Universal Robots PolyScope program: reciprocal_full.urp

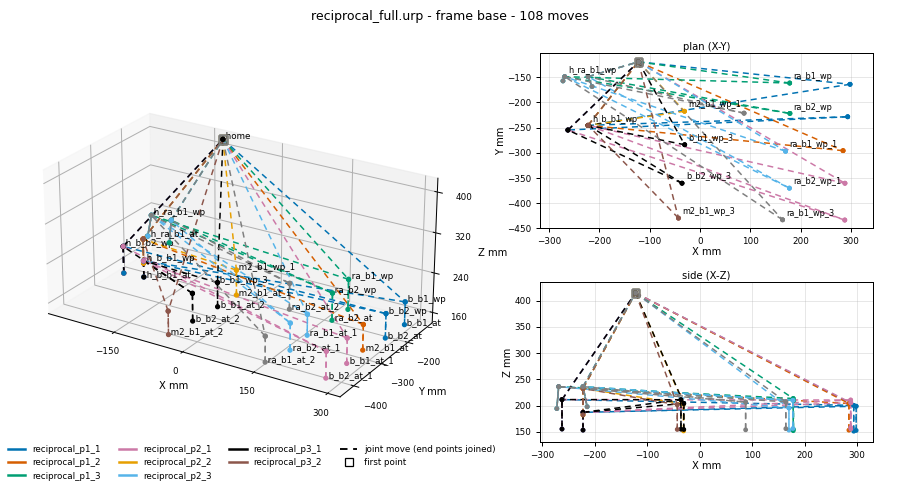
[picture p0: tool path of reciprocal_full.urp in frame base, 108 of 108 moves have a stored position in this frame; points joined in program order, loops and branches not executed]
Program reciprocal_full (installation=default directory=/programs/ITER createdIn=5.3.1.64192 lastSavedIn=5.3.1.64192 robotSerialNumber=20195300365)
Calibrated DH parameters: a=[-0.000093, -0.190649, -0.212673, 0.000091, -0.000205, 0]; d=[0.151591, 44.061648, -42.488068, -1.442789, 0.085322, 0.091911]; alpha=[1.570082, -0.003447, 0.007513, 1.572293, -1.571904, 0]; deltaTheta=[0, -0.672656, 0.728185, -0.055522, 0.000005, 0]
Robot Program (runOnlyOnce=true)
  Call reciprocal_p1_1
  Popup Message (haltProgram=false message=interaction inputType=Text)
  Call reciprocal_p1_2
  Popup Message (haltProgram=false message=interaction inputType=Text)
  Call reciprocal_p1_3
  Popup Message (haltProgram=false message=interaction inputType=Text)
  Call reciprocal_p2_1
  Popup Message (haltProgram=false message=interaction inputType=Text)
  Call reciprocal_p2_2
  Popup Message (haltProgram=false message=interaction inputType=Text)
  Call reciprocal_p2_3
  Popup Message (haltProgram=false message=interaction inputType=Text)
  Call reciprocal_p3_1
  Popup Message (haltProgram=false message=interaction inputType=Text)
  Call reciprocal_p3_2
  Popup Message (haltProgram=false message=interaction inputType=Text)
  Call reciprocal_p3_3
SubProgram -> reciprocal_p3_3
SubProgram -> reciprocal_p3_2
SubProgram -> reciprocal_p3_1
SubProgram -> reciprocal_p2_3
SubProgram -> reciprocal_p2_2
SubProgram -> reciprocal_p2_1
SubProgram -> reciprocal_p1_3
SubProgram -> reciprocal_p1_2
SubProgram -> reciprocal_p1_1
SubProgram reciprocal_p1_1 (keepSynchronizedWithDisk=true trackProgramExecution=false) programFile=/programs/ITER/reciprocal_p1_1.urp
  URCap Gripper Activate (Robotiq_Grippers, Robotiq Inc.) dataModel(ResetAndActivateKey=false)
  URCap Gripper (Robotiq_Grippers, Robotiq Inc.) dataModel(position=50.0, force=100.0, speed=100.0, positionInDouble=50.0, forceInDouble=100.0, speedInDouble=100.0, slaveIds=[9], blocking=true)
  MoveJ speed 60 deg/s, acceleration 80 deg/s^2 (useActiveTCP=true) feature=Base
    Waypoint home: TCP in base x=-122.15 y=-119.32 z=414.454 mm, rx=2.2563 ry=2.1459 rz=-0.0481 rad; joints [-85.681, -56.776, -79.802, -131.025, 89.944, -262.833] deg
  Folder Base
    MoveJ speed 60 deg/s, acceleration 80 deg/s^2 (useActiveTCP=true) feature=Base
      Waypoint b_b1_wp: TCP in base x=297.989 y=-163.874 z=198.695 mm, rx=2.2416 ry=2.1933 rz=-0.0875 rad; joints [-5.657, -99.775, -108.03, -64.017, 87.69, -183.98] deg
      Waypoint b_b1_at: TCP in base x=297.98 y=-163.89 z=152.63 mm, rx=2.2418 ry=2.1932 rz=-0.0874 rad; joints [-5.678, -106.278, -114.473, -51.073, 87.63, -183.927] deg
      URCap Gripper (Robotiq_Grippers, Robotiq Inc.) dataModel(position=100.0, force=100.0, speed=100.0, positionInDouble=100.0, forceInDouble=100.0, speedInDouble=100.0, slaveIds=[9], blocking=true)
      Waypoint b_b1_wp: TCP in base x=297.989 y=-163.874 z=198.695 mm, rx=2.2416 ry=2.1933 rz=-0.0875 rad; joints [-5.657, -99.775, -108.03, -64.017, 87.69, -183.98] deg
      Waypoint h_b_b1_wp: TCP in base x=-222.187 y=-245.349 z=187.06 mm, rx=-3.1315 ry=0.0204 rz=0.0123 rad; joints [-108.957, -99.116, -113.081, -58.146, 89.665, -197.782] deg
      Waypoint h_b_b1_at: TCP in base x=-222.188 y=-245.348 z=153.24 mm, rx=-3.1314 ry=0.0204 rz=0.0122 rad; joints [-108.969, -104.391, -117.643, -48.312, 89.612, -197.745] deg
      URCap Gripper (Robotiq_Grippers, Robotiq Inc.) dataModel(position=50.0, force=100.0, speed=100.0, positionInDouble=50.0, forceInDouble=100.0, speedInDouble=100.0, slaveIds=[9], blocking=true)
      Waypoint h_b_b1_wp: TCP in base x=-222.187 y=-245.349 z=187.06 mm, rx=-3.1315 ry=0.0204 rz=0.0123 rad; joints [-108.957, -99.116, -113.081, -58.146, 89.665, -197.782] deg
    MoveJ speed 60 deg/s, acceleration 80 deg/s^2 (useActiveTCP=true) feature=Base
      Waypoint b_b2_wp: TCP in base x=293.357 y=-228.364 z=200.348 mm, rx=2.2516 ry=2.1757 rz=-0.0473 rad; joints [-17.02, -106.79, -99.111, -64.372, 88.479, -194.689] deg
      Waypoint b_b2_at: TCP in base x=293.371 y=-228.346 z=151.163 mm, rx=2.2516 ry=2.1757 rz=-0.0473 rad; joints [-17.033, -113.072, -105.562, -51.642, 88.423, -194.639] deg
      URCap Gripper (Robotiq_Grippers, Robotiq Inc.) dataModel(position=100.0, force=100.0, speed=100.0, positionInDouble=100.0, forceInDouble=100.0, speedInDouble=100.0, slaveIds=[9], blocking=true)
      Waypoint b_b2_wp: TCP in base x=293.357 y=-228.364 z=200.348 mm, rx=2.2516 ry=2.1757 rz=-0.0473 rad; joints [-17.02, -106.79, -99.111, -64.372, 88.479, -194.689] deg
      Waypoint h_b_b2_wp: TCP in base x=-262.196 y=-254.726 z=211.351 mm, rx=-3.0605 ry=0.0443 rz=-0.0223 rad; joints [-114.749, -105.359, -96.042, -73.109, 89.199, -202.734] deg
      Waypoint h_b_b2_at: TCP in base x=-262.208 y=-254.718 z=155.33 mm, rx=-3.0605 ry=0.0443 rz=-0.0223 rad; joints [-114.774, -111.736, -104.192, -58.581, 89.146, -202.674] deg
      URCap Gripper (Robotiq_Grippers, Robotiq Inc.) dataModel(position=50.0, force=100.0, speed=100.0, positionInDouble=50.0, forceInDouble=100.0, speedInDouble=100.0, slaveIds=[9], blocking=true)
      Waypoint h_b_b2_wp: TCP in base x=-262.196 y=-254.726 z=211.351 mm, rx=-3.0605 ry=0.0443 rz=-0.0223 rad; joints [-114.749, -105.359, -96.042, -73.109, 89.199, -202.734] deg
  MoveJ speed 60 deg/s, acceleration 80 deg/s^2 (useActiveTCP=true) feature=Base
    Waypoint home: TCP in base x=-122.15 y=-119.32 z=414.454 mm, rx=2.2563 ry=2.1459 rz=-0.0481 rad; joints [-85.681, -56.776, -79.802, -131.025, 89.944, -262.833] deg
SubProgram reciprocal_p1_2 (keepSynchronizedWithDisk=true trackProgramExecution=false) programFile=/programs/ITER/reciprocal_p1_2.urp
  URCap Gripper Activate (Robotiq_Grippers, Robotiq Inc.) dataModel(ResetAndActivateKey=false)
  URCap Gripper (Robotiq_Grippers, Robotiq Inc.) dataModel(position=50.0, force=100.0, speed=100.0, positionInDouble=50.0, forceInDouble=100.0, speedInDouble=100.0, slaveIds=[9], blocking=true)
  MoveJ speed 60 deg/s, acceleration 80 deg/s^2 (useActiveTCP=true) feature=Base
    Waypoint home: TCP in base x=-122.15 y=-119.32 z=414.454 mm, rx=2.2563 ry=2.1459 rz=-0.0481 rad; joints [-85.681, -56.776, -79.802, -131.025, 89.944, -262.833] deg
  Folder Mid_2
    MoveJ speed 60 deg/s, acceleration 80 deg/s^2 (useActiveTCP=true) feature=Base
      Waypoint m2_b1_wp: TCP in base x=284.16 y=-295.685 z=203.947 mm, rx=2.2476 ry=2.1381 rz=-0.0269 rad; joints [-27.296, -114.823, -87.386, -65.934, 88.586, -204.141] deg
      Waypoint m2_b1_at: TCP in base x=284.146 y=-295.69 z=153.108 mm, rx=2.2477 ry=2.1381 rz=-0.0269 rad; joints [-27.314, -120.451, -93.885, -53.812, 88.539, -204.094] deg
      URCap Gripper (Robotiq_Grippers, Robotiq Inc.) dataModel(position=100.0, force=100.0, speed=100.0, positionInDouble=100.0, forceInDouble=100.0, speedInDouble=100.0, slaveIds=[9], blocking=true)
      Waypoint m2_b1_wp: TCP in base x=284.16 y=-295.685 z=203.947 mm, rx=2.2476 ry=2.1381 rz=-0.0269 rad; joints [-27.296, -114.823, -87.386, -65.934, 88.586, -204.141] deg
      Waypoint h_m2_b1_wp: TCP in base x=-222.193 y=-245.34 z=232.403 mm, rx=-3.1314 ry=0.0205 rz=0.0123 rad; joints [-108.936, -94.247, -105.13, -70.966, 89.712, -197.837] deg
      Waypoint h_m2_b1_at: TCP in base x=-222.194 y=-245.343 z=182.32 mm, rx=-3.1314 ry=0.0205 rz=0.0122 rad; joints [-108.96, -99.771, -113.792, -56.782, 89.658, -197.776] deg
      URCap Gripper (Robotiq_Grippers, Robotiq Inc.) dataModel(position=50.0, force=100.0, speed=100.0, positionInDouble=50.0, forceInDouble=100.0, speedInDouble=100.0, slaveIds=[9], blocking=true)
      Waypoint h_m2_b1_wp: TCP in base x=-222.193 y=-245.34 z=232.403 mm, rx=-3.1314 ry=0.0205 rz=0.0123 rad; joints [-108.936, -94.247, -105.13, -70.966, 89.712, -197.837] deg
  MoveJ speed 60 deg/s, acceleration 80 deg/s^2 (useActiveTCP=true) feature=Base
    Waypoint home: TCP in base x=-122.15 y=-119.32 z=414.454 mm, rx=2.2563 ry=2.1459 rz=-0.0481 rad; joints [-85.681, -56.776, -79.802, -131.025, 89.944, -262.833] deg
SubProgram reciprocal_p1_3 (keepSynchronizedWithDisk=true trackProgramExecution=false) programFile=/programs/ITER/reciprocal_p1_3.urp
  URCap Gripper Activate (Robotiq_Grippers, Robotiq Inc.) dataModel(ResetAndActivateKey=false)
  URCap Gripper (Robotiq_Grippers, Robotiq Inc.) dataModel(position=50.0, force=100.0, speed=100.0, positionInDouble=50.0, forceInDouble=100.0, speedInDouble=100.0, slaveIds=[9], blocking=true)
  MoveJ speed 60 deg/s, acceleration 80 deg/s^2 (useActiveTCP=true) feature=Base
    Waypoint home: TCP in base x=-122.15 y=-119.32 z=414.454 mm, rx=2.2563 ry=2.1459 rz=-0.0481 rad; joints [-85.681, -56.776, -79.802, -131.025, 89.944, -262.833] deg
  Folder Roof_A
    MoveJ speed 60 deg/s, acceleration 80 deg/s^2 (useActiveTCP=true) feature=Base
      Waypoint ra_b1_wp: TCP in base x=178.147 y=-161.416 z=213.493 mm, rx=2.2107 ry=2.1864 rz=-0.0129 rad; joints [-8.931, -69.528, -131.792, -67.419, 88.9, -187.899] deg
      Waypoint ra_b1_at: TCP in base x=178.14 y=-161.425 z=152.15 mm, rx=2.2108 ry=2.1863 rz=-0.013 rad; joints [-8.971, -81.208, -143.947, -43.587, 88.771, -187.8] deg
      URCap Gripper (Robotiq_Grippers, Robotiq Inc.) dataModel(position=100.0, force=100.0, speed=100.0, positionInDouble=100.0, forceInDouble=100.0, speedInDouble=100.0, slaveIds=[9], blocking=true)
      Waypoint ra_b1_wp: TCP in base x=178.147 y=-161.416 z=213.493 mm, rx=2.2107 ry=2.1864 rz=-0.0129 rad; joints [-8.931, -69.528, -131.792, -67.419, 88.9, -187.899] deg
      Waypoint h_ra_b1_wp: TCP in base x=-268.55 y=-148.787 z=236.04 mm, rx=2.7608 ry=-0.1306 rz=0.0749 rad; joints [-131.096, -88.368, -118.927, -47.1, 105.838, -213.026] deg
      Waypoint h_ra_b1_at: TCP in base x=-272.048 y=-157.193 z=194.251 mm, rx=2.7928 ry=-0.086 rz=0.1068 rad; joints [-130.55, -96.287, -122.586, -37.872, 105.802, -214.66] deg
      URCap Gripper (Robotiq_Grippers, Robotiq Inc.) dataModel(position=50.0, force=100.0, speed=100.0, positionInDouble=50.0, forceInDouble=100.0, speedInDouble=100.0, slaveIds=[9], blocking=true)
      Waypoint h_ra_b1_wp: TCP in base x=-268.55 y=-148.787 z=236.04 mm, rx=2.7608 ry=-0.1306 rz=0.0749 rad; joints [-131.096, -88.368, -118.927, -47.1, 105.838, -213.026] deg
    MoveJ speed 60 deg/s, acceleration 80 deg/s^2 (useActiveTCP=true) feature=Base
      Waypoint ra_b2_wp: TCP in base x=178.587 y=-221.707 z=209.682 mm, rx=2.2093 ry=2.1872 rz=-0.0611 rad; joints [-23.097, -83.646, -122.705, -62.748, 87.545, -202.118] deg
      Waypoint ra_b2_at: TCP in base x=178.563 y=-221.705 z=154.679 mm, rx=2.2094 ry=2.1872 rz=-0.0612 rad; joints [-23.123, -93.044, -131.897, -44.166, 87.443, -202.046] deg
      URCap Gripper (Robotiq_Grippers, Robotiq Inc.) dataModel(position=100.0, force=100.0, speed=100.0, positionInDouble=100.0, forceInDouble=100.0, speedInDouble=100.0, slaveIds=[9], blocking=true)
      Waypoint ra_b2_wp: TCP in base x=178.587 y=-221.707 z=209.682 mm, rx=2.2093 ry=2.1872 rz=-0.0611 rad; joints [-23.097, -83.646, -122.705, -62.748, 87.545, -202.118] deg
      Waypoint h_ra_b2_wp: TCP in base x=-222.173 y=-148.778 z=236.048 mm, rx=2.7617 ry=-0.0717 rz=0.0011 rad; joints [-121.367, -76.176, -130.557, -44.074, 100.878, -206.047] deg
      Waypoint h_ra_b2_at: TCP in base x=-214.314 y=-168.312 z=197.793 mm, rx=2.8721 ry=-0.0559 rz=-0.0607 rad; joints [-115.061, -82.329, -135.249, -37.27, 94.17, -201.737] deg
      URCap Gripper (Robotiq_Grippers, Robotiq Inc.) dataModel(position=50.0, force=100.0, speed=100.0, positionInDouble=50.0, forceInDouble=100.0, speedInDouble=100.0, slaveIds=[9], blocking=true)
      Waypoint h_ra_b2_wp: TCP in base x=-222.173 y=-148.778 z=236.048 mm, rx=2.7617 ry=-0.0717 rz=0.0011 rad; joints [-121.367, -76.176, -130.557, -44.074, 100.878, -206.047] deg
  MoveJ speed 60 deg/s, acceleration 80 deg/s^2 (useActiveTCP=true) feature=Base
    Waypoint home: TCP in base x=-122.15 y=-119.32 z=414.454 mm, rx=2.2563 ry=2.1459 rz=-0.0481 rad; joints [-85.681, -56.776, -79.802, -131.025, 89.944, -262.833] deg
SubProgram reciprocal_p2_1 (keepSynchronizedWithDisk=true trackProgramExecution=false) programFile=/programs/ITER/reciprocal_p2_1.urp
  URCap Gripper Activate (Robotiq_Grippers, Robotiq Inc.) dataModel(ResetAndActivateKey=false)
  URCap Gripper (Robotiq_Grippers, Robotiq Inc.) dataModel(position=50.0, force=100.0, speed=100.0, positionInDouble=50.0, forceInDouble=100.0, speedInDouble=100.0, slaveIds=[9], blocking=true)
  MoveJ speed 60 deg/s, acceleration 80 deg/s^2 (useActiveTCP=true) feature=Base
    Waypoint home: TCP in base x=-122.15 y=-119.32 z=414.454 mm, rx=2.2563 ry=2.1459 rz=-0.0481 rad; joints [-85.681, -56.776, -79.802, -131.025, 89.944, -262.833] deg
  Folder Base
    MoveJ speed 60 deg/s, acceleration 80 deg/s^2 (useActiveTCP=true) feature=Base
      Waypoint b_b1_wp_1: TCP in base x=287.856 y=-360.368 z=205.358 mm, rx=2.2407 ry=2.1786 rz=-0.0803 rad; joints [-34.358, -127.348, -66.069, -76.253, 87.212, -212.545] deg
      Waypoint b_b1_at_1: TCP in base x=287.864 y=-360.357 z=155.443 mm, rx=2.2407 ry=2.1786 rz=-0.0802 rad; joints [-34.375, -131.385, -73.13, -65.157, 87.19, -212.499] deg
      URCap Gripper (Robotiq_Grippers, Robotiq Inc.) dataModel(position=100.0, force=100.0, speed=100.0, positionInDouble=100.0, forceInDouble=100.0, speedInDouble=100.0, slaveIds=[9], blocking=true)
      Waypoint b_b1_wp_2: TCP in base x=287.856 y=-360.368 z=205.358 mm, rx=2.2407 ry=2.1786 rz=-0.0803 rad; joints [-34.358, -127.348, -66.069, -76.253, 87.212, -212.545] deg
      Waypoint h_b_b1_wp: TCP in base x=-222.187 y=-245.349 z=187.06 mm, rx=-3.1315 ry=0.0204 rz=0.0123 rad; joints [-108.957, -99.116, -113.081, -58.146, 89.665, -197.782] deg
      Waypoint h_b_b1_at: TCP in base x=-222.188 y=-245.348 z=153.24 mm, rx=-3.1314 ry=0.0204 rz=0.0122 rad; joints [-108.969, -104.391, -117.643, -48.312, 89.612, -197.745] deg
      URCap Gripper (Robotiq_Grippers, Robotiq Inc.) dataModel(position=50.0, force=100.0, speed=100.0, positionInDouble=50.0, forceInDouble=100.0, speedInDouble=100.0, slaveIds=[9], blocking=true)
      Waypoint h_b_b1_wp: TCP in base x=-222.187 y=-245.349 z=187.06 mm, rx=-3.1315 ry=0.0204 rz=0.0123 rad; joints [-108.957, -99.116, -113.081, -58.146, 89.665, -197.782] deg
    MoveJ speed 60 deg/s, acceleration 80 deg/s^2 (useActiveTCP=true) feature=Base
      Waypoint b_b2_wp_1: TCP in base x=287.521 y=-433.433 z=210.514 mm, rx=2.2195 ry=2.211 rz=-0.063 rad; joints [-41.44, -147.038, -28.419, -94.163, 87.942, -221.217] deg
      Waypoint b_b2_at_1: TCP in base x=287.518 y=-433.44 z=158.432 mm, rx=2.2196 ry=2.211 rz=-0.063 rad; joints [-41.471, -147.777, -41.016, -80.833, 87.944, -221.148] deg
      URCap Gripper (Robotiq_Grippers, Robotiq Inc.) dataModel(position=100.0, force=100.0, speed=100.0, positionInDouble=100.0, forceInDouble=100.0, speedInDouble=100.0, slaveIds=[9], blocking=true)
      Waypoint b_b2_wp_2: TCP in base x=287.521 y=-433.433 z=210.514 mm, rx=2.2195 ry=2.211 rz=-0.063 rad; joints [-41.44, -147.038, -28.419, -94.163, 87.942, -221.217] deg
      Waypoint h_b_b2_wp: TCP in base x=-262.196 y=-254.726 z=211.351 mm, rx=-3.0605 ry=0.0443 rz=-0.0223 rad; joints [-114.749, -105.359, -96.042, -73.109, 89.199, -202.734] deg
      Waypoint h_b_b2_at: TCP in base x=-262.208 y=-254.718 z=155.33 mm, rx=-3.0605 ry=0.0443 rz=-0.0223 rad; joints [-114.774, -111.736, -104.192, -58.581, 89.146, -202.674] deg
      URCap Gripper (Robotiq_Grippers, Robotiq Inc.) dataModel(position=50.0, force=100.0, speed=100.0, positionInDouble=50.0, forceInDouble=100.0, speedInDouble=100.0, slaveIds=[9], blocking=true)
      Waypoint h_b_b2_wp: TCP in base x=-262.196 y=-254.726 z=211.351 mm, rx=-3.0605 ry=0.0443 rz=-0.0223 rad; joints [-114.749, -105.359, -96.042, -73.109, 89.199, -202.734] deg
  MoveJ speed 60 deg/s, acceleration 80 deg/s^2 (useActiveTCP=true) feature=Base
    Waypoint home: TCP in base x=-122.15 y=-119.32 z=414.454 mm, rx=2.2563 ry=2.1459 rz=-0.0481 rad; joints [-85.681, -56.776, -79.802, -131.025, 89.944, -262.833] deg
SubProgram reciprocal_p2_2 (keepSynchronizedWithDisk=true trackProgramExecution=false) programFile=/programs/ITER/reciprocal_p2_2.urp
  URCap Gripper Activate (Robotiq_Grippers, Robotiq Inc.) dataModel(ResetAndActivateKey=false)
  URCap Gripper (Robotiq_Grippers, Robotiq Inc.) dataModel(position=50.0, force=100.0, speed=100.0, positionInDouble=50.0, forceInDouble=100.0, speedInDouble=100.0, slaveIds=[9], blocking=true)
  MoveJ speed 60 deg/s, acceleration 80 deg/s^2 (useActiveTCP=true) feature=Base
    Waypoint home: TCP in base x=-122.15 y=-119.32 z=414.454 mm, rx=2.2563 ry=2.1459 rz=-0.0481 rad; joints [-85.681, -56.776, -79.802, -131.025, 89.944, -262.833] deg
  Folder Mid_2
    MoveJ speed 60 deg/s, acceleration 80 deg/s^2 (useActiveTCP=true) feature=Base
      Waypoint m2_b1_wp_1: TCP in base x=-30.704 y=-217.422 z=203.363 mm, rx=-2.2397 ry=-2.1922 rz=0.0003 rad; joints [-61.845, -63.917, -136.913, -69.519, 90.279, -240.21] deg
      Waypoint m2_b1_at_1: TCP in base x=-30.716 y=-217.427 z=151.677 mm, rx=-2.2397 ry=-2.1922 rz=0.0003 rad; joints [-61.887, -74.21, -147.891, -48.249, 90.169, -240.122] deg
      URCap Gripper (Robotiq_Grippers, Robotiq Inc.) dataModel(position=100.0, force=100.0, speed=100.0, positionInDouble=100.0, forceInDouble=100.0, speedInDouble=100.0, slaveIds=[9], blocking=true)
      Waypoint m2_b1_wp_2: TCP in base x=-30.704 y=-217.422 z=203.363 mm, rx=-2.2397 ry=-2.1922 rz=0.0003 rad; joints [-61.845, -63.917, -136.913, -69.519, 90.279, -240.21] deg
      Waypoint h_m2_b1_wp: TCP in base x=-222.193 y=-245.34 z=232.403 mm, rx=-3.1314 ry=0.0205 rz=0.0123 rad; joints [-108.936, -94.247, -105.13, -70.966, 89.712, -197.837] deg
      Waypoint h_m2_b1_at: TCP in base x=-222.194 y=-245.343 z=182.32 mm, rx=-3.1314 ry=0.0205 rz=0.0122 rad; joints [-108.96, -99.771, -113.792, -56.782, 89.658, -197.776] deg
      URCap Gripper (Robotiq_Grippers, Robotiq Inc.) dataModel(position=50.0, force=100.0, speed=100.0, positionInDouble=50.0, forceInDouble=100.0, speedInDouble=100.0, slaveIds=[9], blocking=true)
      Waypoint h_m2_b1_wp: TCP in base x=-222.193 y=-245.34 z=232.403 mm, rx=-3.1314 ry=0.0205 rz=0.0123 rad; joints [-108.936, -94.247, -105.13, -70.966, 89.712, -197.837] deg
  MoveJ speed 60 deg/s, acceleration 80 deg/s^2 (useActiveTCP=true) feature=Base
    Waypoint home: TCP in base x=-122.15 y=-119.32 z=414.454 mm, rx=2.2563 ry=2.1459 rz=-0.0481 rad; joints [-85.681, -56.776, -79.802, -131.025, 89.944, -262.833] deg
SubProgram reciprocal_p2_3 (keepSynchronizedWithDisk=true trackProgramExecution=false) programFile=/programs/ITER/reciprocal_p2_3.urp
  URCap Gripper Activate (Robotiq_Grippers, Robotiq Inc.) dataModel(ResetAndActivateKey=false)
  URCap Gripper (Robotiq_Grippers, Robotiq Inc.) dataModel(position=50.0, force=100.0, speed=100.0, positionInDouble=50.0, forceInDouble=100.0, speedInDouble=100.0, slaveIds=[9], blocking=true)
  MoveJ speed 60 deg/s, acceleration 80 deg/s^2 (useActiveTCP=true) feature=Base
    Waypoint home: TCP in base x=-122.15 y=-119.32 z=414.454 mm, rx=2.2563 ry=2.1459 rz=-0.0481 rad; joints [-85.681, -56.776, -79.802, -131.025, 89.944, -262.833] deg
  Folder Roof_A
    MoveJ speed 60 deg/s, acceleration 80 deg/s^2 (useActiveTCP=true) feature=Base
      Waypoint ra_b1_wp_1: TCP in base x=169.973 y=-296.809 z=195.434 mm, rx=2.2324 ry=2.1892 rz=0.039 rad; joints [-38.336, -100.686, -109.203, -59.029, 91.581, -216.79] deg
      Waypoint ra_b1_at_1: TCP in base x=169.98 y=-296.801 z=153.211 mm, rx=2.2324 ry=2.1893 rz=0.0391 rad; joints [-38.349, -106.915, -114.861, -47.14, 91.523, -216.748] deg
      URCap Gripper (Robotiq_Grippers, Robotiq Inc.) dataModel(position=100.0, force=100.0, speed=100.0, positionInDouble=100.0, forceInDouble=100.0, speedInDouble=100.0, slaveIds=[9], blocking=true)
      Waypoint ra_b1_wp_2: TCP in base x=169.973 y=-296.809 z=195.434 mm, rx=2.2324 ry=2.1892 rz=0.039 rad; joints [-38.336, -100.686, -109.203, -59.029, 91.581, -216.79] deg
      Waypoint h_ra_b1_wp: TCP in base x=-268.55 y=-148.787 z=236.04 mm, rx=2.7608 ry=-0.1306 rz=0.0749 rad; joints [-131.096, -88.368, -118.927, -47.1, 105.838, -213.026] deg
      Waypoint h_ra_b1_at: TCP in base x=-272.048 y=-157.193 z=194.251 mm, rx=2.7928 ry=-0.086 rz=0.1068 rad; joints [-130.55, -96.287, -122.586, -37.872, 105.802, -214.66] deg
      URCap Gripper (Robotiq_Grippers, Robotiq Inc.) dataModel(position=50.0, force=100.0, speed=100.0, positionInDouble=50.0, forceInDouble=100.0, speedInDouble=100.0, slaveIds=[9], blocking=true)
      Waypoint h_ra_b1_wp: TCP in base x=-268.55 y=-148.787 z=236.04 mm, rx=2.7608 ry=-0.1306 rz=0.0749 rad; joints [-131.096, -88.368, -118.927, -47.1, 105.838, -213.026] deg
    MoveJ speed 60 deg/s, acceleration 80 deg/s^2 (useActiveTCP=true) feature=Base
      Waypoint ra_b2_wp_1: TCP in base x=177.575 y=-370.13 z=209.996 mm, rx=-2.2477 ry=-2.162 rz=0.0032 rad; joints [-45.905, -115.327, -83.545, -72.376, 90.171, -223.395] deg
      Waypoint ra_b2_at_1: TCP in base x=177.559 y=-370.143 z=156.36 mm, rx=-2.2478 ry=-2.1619 rz=0.0031 rad; joints [-45.928, -120.68, -90.962, -59.606, 90.129, -223.34] deg
      URCap Gripper (Robotiq_Grippers, Robotiq Inc.) dataModel(position=100.0, force=100.0, speed=100.0, positionInDouble=100.0, forceInDouble=100.0, speedInDouble=100.0, slaveIds=[9], blocking=true)
      Waypoint ra_b2_wp_2: TCP in base x=177.575 y=-370.13 z=209.996 mm, rx=-2.2477 ry=-2.162 rz=0.0032 rad; joints [-45.905, -115.327, -83.545, -72.376, 90.171, -223.395] deg
      Waypoint h_ra_b2_wp: TCP in base x=-222.173 y=-148.778 z=236.048 mm, rx=2.7617 ry=-0.0717 rz=0.0011 rad; joints [-121.367, -76.176, -130.557, -44.074, 100.878, -206.047] deg
      Waypoint h_ra_b2_at: TCP in base x=-214.314 y=-168.312 z=197.793 mm, rx=2.8721 ry=-0.0559 rz=-0.0607 rad; joints [-115.061, -82.329, -135.249, -37.27, 94.17, -201.737] deg
      URCap Gripper (Robotiq_Grippers, Robotiq Inc.) dataModel(position=50.0, force=100.0, speed=100.0, positionInDouble=50.0, forceInDouble=100.0, speedInDouble=100.0, slaveIds=[9], blocking=true)
      Waypoint h_ra_b2_wp: TCP in base x=-222.173 y=-148.778 z=236.048 mm, rx=2.7617 ry=-0.0717 rz=0.0011 rad; joints [-121.367, -76.176, -130.557, -44.074, 100.878, -206.047] deg
  MoveJ speed 60 deg/s, acceleration 80 deg/s^2 (useActiveTCP=true) feature=Base
    Waypoint home: TCP in base x=-122.15 y=-119.32 z=414.454 mm, rx=2.2563 ry=2.1459 rz=-0.0481 rad; joints [-85.681, -56.776, -79.802, -131.025, 89.944, -262.833] deg
SubProgram reciprocal_p3_1 (keepSynchronizedWithDisk=true trackProgramExecution=false) programFile=/programs/ITER/reciprocal_p3_1.urp
  URCap Gripper Activate (Robotiq_Grippers, Robotiq Inc.) dataModel(ResetAndActivateKey=false)
  URCap Gripper (Robotiq_Grippers, Robotiq Inc.) dataModel(position=50.0, force=100.0, speed=100.0, positionInDouble=50.0, forceInDouble=100.0, speedInDouble=100.0, slaveIds=[9], blocking=true)
  MoveJ speed 60 deg/s, acceleration 80 deg/s^2 (useActiveTCP=true) feature=Base
    Waypoint home: TCP in base x=-122.15 y=-119.32 z=414.454 mm, rx=2.2563 ry=2.1459 rz=-0.0481 rad; joints [-85.681, -56.776, -79.802, -131.025, 89.944, -262.833] deg
  Folder Base
    MoveJ speed 60 deg/s, acceleration 80 deg/s^2 (useActiveTCP=true) feature=Base
      Waypoint b_b1_wp_3: TCP in base x=-30.305 y=-283.938 z=204.008 mm, rx=-2.2165 ry=-2.2166 rz=0.0302 rad; joints [-68.72, -85.09, -122.783, -61.983, 89.153, -248.292] deg
      Waypoint b_b1_at_2: TCP in base x=-30.308 y=-283.929 z=154.464 mm, rx=-2.2165 ry=-2.2166 rz=0.0302 rad; joints [-68.742, -93.618, -130.893, -45.349, 89.063, -248.228] deg
      URCap Gripper (Robotiq_Grippers, Robotiq Inc.) dataModel(position=100.0, force=100.0, speed=100.0, positionInDouble=100.0, forceInDouble=100.0, speedInDouble=100.0, slaveIds=[9], blocking=true)
      Waypoint b_b1_wp_4: TCP in base x=-30.305 y=-283.938 z=204.008 mm, rx=-2.2165 ry=-2.2166 rz=0.0302 rad; joints [-68.72, -85.09, -122.783, -61.983, 89.153, -248.292] deg
      Waypoint h_b_b1_wp: TCP in base x=-222.187 y=-245.349 z=187.06 mm, rx=-3.1315 ry=0.0204 rz=0.0123 rad; joints [-108.957, -99.116, -113.081, -58.146, 89.665, -197.782] deg
      Waypoint h_b_b1_at: TCP in base x=-222.188 y=-245.348 z=153.24 mm, rx=-3.1314 ry=0.0204 rz=0.0122 rad; joints [-108.969, -104.391, -117.643, -48.312, 89.612, -197.745] deg
      URCap Gripper (Robotiq_Grippers, Robotiq Inc.) dataModel(position=50.0, force=100.0, speed=100.0, positionInDouble=50.0, forceInDouble=100.0, speedInDouble=100.0, slaveIds=[9], blocking=true)
      Waypoint h_b_b1_wp: TCP in base x=-222.187 y=-245.349 z=187.06 mm, rx=-3.1315 ry=0.0204 rz=0.0123 rad; joints [-108.957, -99.116, -113.081, -58.146, 89.665, -197.782] deg
    MoveJ speed 60 deg/s, acceleration 80 deg/s^2 (useActiveTCP=true) feature=Base
      Waypoint b_b2_wp_3: TCP in base x=-35.668 y=-360.302 z=211.088 mm, rx=-2.2184 ry=-2.2071 rz=-0.0146 rad; joints [-74.709, -103.844, -99.62, -67.347, 90.409, -254.067] deg
      Waypoint b_b2_at_2: TCP in base x=-35.691 y=-360.3 z=154.951 mm, rx=-2.2183 ry=-2.2071 rz=-0.0145 rad; joints [-74.732, -110.771, -107.538, -52.502, 90.342, -254.01] deg
      URCap Gripper (Robotiq_Grippers, Robotiq Inc.) dataModel(position=100.0, force=100.0, speed=100.0, positionInDouble=100.0, forceInDouble=100.0, speedInDouble=100.0, slaveIds=[9], blocking=true)
      Waypoint b_b2_wp_4: TCP in base x=-35.668 y=-360.302 z=211.088 mm, rx=-2.2184 ry=-2.2071 rz=-0.0146 rad; joints [-74.709, -103.844, -99.62, -67.347, 90.409, -254.067] deg
      Waypoint h_b_b2_wp: TCP in base x=-262.196 y=-254.726 z=211.351 mm, rx=-3.0605 ry=0.0443 rz=-0.0223 rad; joints [-114.749, -105.359, -96.042, -73.109, 89.199, -202.734] deg
      Waypoint h_b_b2_at: TCP in base x=-262.208 y=-254.718 z=155.33 mm, rx=-3.0605 ry=0.0443 rz=-0.0223 rad; joints [-114.774, -111.736, -104.192, -58.581, 89.146, -202.674] deg
      URCap Gripper (Robotiq_Grippers, Robotiq Inc.) dataModel(position=50.0, force=100.0, speed=100.0, positionInDouble=50.0, forceInDouble=100.0, speedInDouble=100.0, slaveIds=[9], blocking=true)
      Waypoint h_b_b2_wp: TCP in base x=-262.196 y=-254.726 z=211.351 mm, rx=-3.0605 ry=0.0443 rz=-0.0223 rad; joints [-114.749, -105.359, -96.042, -73.109, 89.199, -202.734] deg
  MoveJ speed 60 deg/s, acceleration 80 deg/s^2 (useActiveTCP=true) feature=Base
    Waypoint home: TCP in base x=-122.15 y=-119.32 z=414.454 mm, rx=2.2563 ry=2.1459 rz=-0.0481 rad; joints [-85.681, -56.776, -79.802, -131.025, 89.944, -262.833] deg
SubProgram reciprocal_p3_2 (keepSynchronizedWithDisk=true trackProgramExecution=false) programFile=/programs/ITER/reciprocal_p3_2.urp
  URCap Gripper Activate (Robotiq_Grippers, Robotiq Inc.) dataModel(ResetAndActivateKey=false)
  URCap Gripper (Robotiq_Grippers, Robotiq Inc.) dataModel(position=50.0, force=100.0, speed=100.0, positionInDouble=50.0, forceInDouble=100.0, speedInDouble=100.0, slaveIds=[9], blocking=true)
  MoveJ speed 60 deg/s, acceleration 80 deg/s^2 (useActiveTCP=true) feature=Base
    Waypoint home: TCP in base x=-122.15 y=-119.32 z=414.454 mm, rx=2.2563 ry=2.1459 rz=-0.0481 rad; joints [-85.681, -56.776, -79.802, -131.025, 89.944, -262.833] deg
  Folder Mid_2
    MoveJ speed 60 deg/s, acceleration 80 deg/s^2 (useActiveTCP=true) feature=Base
      Waypoint m2_b1_wp_3: TCP in base x=-42.705 y=-429.628 z=201.674 mm, rx=2.2154 ry=2.1777 rz=0.0173 rad; joints [-78.53, -120.549, -78.862, -69.183, 91.892, -257.242] deg
      Waypoint m2_b1_at_2: TCP in base x=-42.72 y=-429.623 z=154.534 mm, rx=2.2155 ry=2.1777 rz=0.0173 rad; joints [-78.548, -125.214, -84.966, -58.413, 91.858, -257.198] deg
      URCap Gripper (Robotiq_Grippers, Robotiq Inc.) dataModel(position=100.0, force=100.0, speed=100.0, positionInDouble=100.0, forceInDouble=100.0, speedInDouble=100.0, slaveIds=[9], blocking=true)
      Waypoint m2_b1_wp_4: TCP in base x=-42.705 y=-429.628 z=201.674 mm, rx=2.2154 ry=2.1777 rz=0.0173 rad; joints [-78.53, -120.549, -78.862, -69.183, 91.892, -257.242] deg
      Waypoint h_m2_b1_wp: TCP in base x=-222.193 y=-245.34 z=232.403 mm, rx=-3.1314 ry=0.0205 rz=0.0123 rad; joints [-108.936, -94.247, -105.13, -70.966, 89.712, -197.837] deg
      Waypoint h_m2_b1_at: TCP in base x=-222.194 y=-245.343 z=182.32 mm, rx=-3.1314 ry=0.0205 rz=0.0122 rad; joints [-108.96, -99.771, -113.792, -56.782, 89.658, -197.776] deg
      URCap Gripper (Robotiq_Grippers, Robotiq Inc.) dataModel(position=50.0, force=100.0, speed=100.0, positionInDouble=50.0, forceInDouble=100.0, speedInDouble=100.0, slaveIds=[9], blocking=true)
      Waypoint h_m2_b1_wp: TCP in base x=-222.193 y=-245.34 z=232.403 mm, rx=-3.1314 ry=0.0205 rz=0.0123 rad; joints [-108.936, -94.247, -105.13, -70.966, 89.712, -197.837] deg
  MoveJ speed 60 deg/s, acceleration 80 deg/s^2 (useActiveTCP=true) feature=Base
    Waypoint home: TCP in base x=-122.15 y=-119.32 z=414.454 mm, rx=2.2563 ry=2.1459 rz=-0.0481 rad; joints [-85.681, -56.776, -79.802, -131.025, 89.944, -262.833] deg
SubProgram reciprocal_p3_3 (keepSynchronizedWithDisk=true trackProgramExecution=false) programFile=/programs/ITER/reciprocal_p3_3.urp
  URCap Gripper Activate (Robotiq_Grippers, Robotiq Inc.) dataModel(ResetAndActivateKey=false)
  URCap Gripper (Robotiq_Grippers, Robotiq Inc.) dataModel(position=50.0, force=100.0, speed=100.0, positionInDouble=50.0, forceInDouble=100.0, speedInDouble=100.0, slaveIds=[9], blocking=true)
  MoveJ speed 60 deg/s, acceleration 80 deg/s^2 (useActiveTCP=true) feature=Base
    Waypoint home: TCP in base x=-122.15 y=-119.32 z=414.454 mm, rx=2.2563 ry=2.1459 rz=-0.0481 rad; joints [-85.681, -56.776, -79.802, -131.025, 89.944, -262.833] deg
  Folder Roof_A
    MoveJ speed 60 deg/s, acceleration 80 deg/s^2 (useActiveTCP=true) feature=Base
      Waypoint ra_b1_wp_3: TCP in base x=164.04 y=-432.993 z=207.005 mm, rx=2.2314 ry=2.1509 rz=0.0059 rad; joints [-53.036, -127.512, -66.191, -73.855, 90.777, -230.696] deg
      Waypoint ra_b1_at_2: TCP in base x=164.049 y=-432.987 z=156.003 mm, rx=2.2314 ry=2.151 rz=0.0059 rad; joints [-53.052, -131.715, -73.279, -62.563, 90.747, -230.647] deg
      URCap Gripper (Robotiq_Grippers, Robotiq Inc.) dataModel(position=100.0, force=100.0, speed=100.0, positionInDouble=100.0, forceInDouble=100.0, speedInDouble=100.0, slaveIds=[9], blocking=true)
      Waypoint ra_b1_wp_4: TCP in base x=164.04 y=-432.993 z=207.005 mm, rx=2.2314 ry=2.1509 rz=0.0059 rad; joints [-53.036, -127.512, -66.191, -73.855, 90.777, -230.696] deg
      Waypoint h_ra_b1_wp: TCP in base x=-268.55 y=-148.787 z=236.04 mm, rx=2.7608 ry=-0.1306 rz=0.0749 rad; joints [-131.096, -88.368, -118.927, -47.1, 105.838, -213.026] deg
      Waypoint h_ra_b1_at: TCP in base x=-272.048 y=-157.193 z=194.251 mm, rx=2.7928 ry=-0.086 rz=0.1068 rad; joints [-130.55, -96.287, -122.586, -37.872, 105.802, -214.66] deg
      URCap Gripper (Robotiq_Grippers, Robotiq Inc.) dataModel(position=50.0, force=100.0, speed=100.0, positionInDouble=50.0, forceInDouble=100.0, speedInDouble=100.0, slaveIds=[9], blocking=true)
      Waypoint h_ra_b1_wp: TCP in base x=-268.55 y=-148.787 z=236.04 mm, rx=2.7608 ry=-0.1306 rz=0.0749 rad; joints [-131.096, -88.368, -118.927, -47.1, 105.838, -213.026] deg
    MoveJ speed 60 deg/s, acceleration 80 deg/s^2 (useActiveTCP=true) feature=Base
      Waypoint ra_b2_wp_3: TCP in base x=87.515 y=-221.249 z=206.702 mm, rx=2.1687 ry=2.2623 rz=-0.0123 rad; joints [-35.23, -70.004, -133.115, -66.455, 89.869, -217.229] deg
      Waypoint ra_b2_at_2: TCP in base x=87.508 y=-221.258 z=153.772 mm, rx=2.1686 ry=2.2623 rz=-0.0124 rad; joints [-35.265, -80.236, -143.583, -45.752, 89.755, -217.149] deg
      URCap Gripper (Robotiq_Grippers, Robotiq Inc.) dataModel(position=100.0, force=100.0, speed=100.0, positionInDouble=100.0, forceInDouble=100.0, speedInDouble=100.0, slaveIds=[9], blocking=true)
      Waypoint ra_b2_wp_4: TCP in base x=87.515 y=-221.249 z=206.702 mm, rx=2.1687 ry=2.2623 rz=-0.0123 rad; joints [-35.23, -70.004, -133.115, -66.455, 89.869, -217.229] deg
      Waypoint h_ra_b2_wp: TCP in base x=-222.173 y=-148.778 z=236.048 mm, rx=2.7617 ry=-0.0717 rz=0.0011 rad; joints [-121.367, -76.176, -130.557, -44.074, 100.878, -206.047] deg
      Waypoint h_ra_b2_at: TCP in base x=-214.314 y=-168.312 z=197.793 mm, rx=2.8721 ry=-0.0559 rz=-0.0607 rad; joints [-115.061, -82.329, -135.249, -37.27, 94.17, -201.737] deg
      URCap Gripper (Robotiq_Grippers, Robotiq Inc.) dataModel(position=50.0, force=100.0, speed=100.0, positionInDouble=50.0, forceInDouble=100.0, speedInDouble=100.0, slaveIds=[9], blocking=true)
      Waypoint h_ra_b2_wp: TCP in base x=-222.173 y=-148.778 z=236.048 mm, rx=2.7617 ry=-0.0717 rz=0.0011 rad; joints [-121.367, -76.176, -130.557, -44.074, 100.878, -206.047] deg
  MoveJ speed 60 deg/s, acceleration 80 deg/s^2 (useActiveTCP=true) feature=Base
    Waypoint home: TCP in base x=-122.15 y=-119.32 z=414.454 mm, rx=2.2563 ry=2.1459 rz=-0.0481 rad; joints [-85.681, -56.776, -79.802, -131.025, 89.944, -262.833] deg
